// TIA Portal project "DaxiExample" (V15.1)

(* hardware
DEVICE "S71500/ET200MP station_1"  S7-1500 station
   slot 0: "Rail_0"  Rack  6ES7 590-1***0-0AA0
   slot 1: "PLC_4"  CPU 1511-1 PN  6ES7 511-1AK02-0AB0  V2.6
      slot 3: "CPU display_1"  6ES7591-1AA00-0AA0
*)

// ===== PLC "PLC_4"  CPU 1511-1 PN =====

VAR_GLOBAL   // PLC tag table "Default tag table"
   "System_Byte" AT %MB1 : Byte;
   "FirstScan" AT %M1.0 : Bool;
   "DiagStatusUpdate" AT %M1.1 : Bool;
   "AlwaysTRUE" AT %M1.2 : Bool;
   "AlwaysFALSE" AT %M1.3 : Bool;
   "Clock_Byte" AT %MB0 : Byte;
   "Clock_10Hz" AT %M0.0 : Bool;
   "Clock_5Hz" AT %M0.1 : Bool;
   "Clock_2.5Hz" AT %M0.2 : Bool;
   "Clock_2Hz" AT %M0.3 : Bool;
   "Clock_1.25Hz" AT %M0.4 : Bool;
   "Clock_1Hz" AT %M0.5 : Bool;
   "Clock_0.625Hz" AT %M0.6 : Bool;
   "Clock_0.5Hz" AT %M0.7 : Bool;
END_VAR

VAR_GLOBAL   // PLC tag table "Tag table_1"
   "send" AT %M10.0 : Bool;
   "recieve" AT %M10.1 : Bool;
END_VAR

VAR_GLOBAL   // PLC tag table "io"
   "input" AT %I0.0 : Bool;
   "output" AT %Q0.0 : Bool;
END_VAR

DATA_BLOCK "Sensor"   // DB1
{ S7_Optimized_Access := 'FALSE' }
VERSION : 0.1
   VAR
      liveBit : Bool;
      S_channel : Array[0..9] of Struct
         value : Real;
         state : USInt;
         error : Bool;
      END_STRUCT;
   END_VAR
BEGIN
END_DATA_BLOCK

DATA_BLOCK "Inputs"   // DB2
{ S7_Optimized_Access := 'FALSE' }
VERSION : 0.1
   VAR
      livebit : Bool;
      I_channel : Array[0..2] of Bool;
   END_VAR
BEGIN
END_DATA_BLOCK

DATA_BLOCK "Outputs"   // DB3
{ S7_Optimized_Access := 'FALSE' }
VERSION : 0.1
   VAR
      livebit : Bool;
      O_channel : Array[0..11] of Bool;
   END_VAR
BEGIN
END_DATA_BLOCK

DATA_BLOCK "Virtual"   // DB4
{ S7_Optimized_Access := 'FALSE' }
VERSION : 0.1
   VAR
      livebit : Bool;
      virt_index : Array[0..31] of UDInt;
   END_VAR
BEGIN
END_DATA_BLOCK

DATA_BLOCK "Ping"   // DB5
{ S7_Optimized_Access := 'FALSE' }
VERSION : 0.1
   VAR
      livebit : Bool;
      ping_index : Array[0..9] of Bool;
   END_VAR
BEGIN
END_DATA_BLOCK

ORGANIZATION_BLOCK "Main"   // OB1, LAD, ProgramCycle
TITLE = "Main Program Sweep (Cycle)"
{ S7_Optimized_Access := 'TRUE' }
VERSION : 0.1
   VAR_INPUT
      Initial_Call : Bool;   // Initial call of this OB
      Remanence : Bool;   // =True, if remanent data are available
   END_VAR
BEGIN
END_ORGANIZATION_BLOCK